(*TERMINAL 880KF1 - EL2008 ************************************************************************)
	qb880KF1_1_SignalToFockeReady								AT %Q* : BOOL; (* 880KF1_1 *)
	qb880KF1_5_SignalToFockeCutOut								AT %Q* : BOOL; (* 880KF1_5 *)
	qb880KF1_2_SignalToFockeRejectOuter							AT %Q* : BOOL; (* 880KF1_2 *)
	qb880KF1_6_SignalToFockeRejectLimitReachedTrigger			AT %Q* : BOOL; (* 880KF1_6 *)
	qb880KF1_3_SignalToFockeDynamicCameraTriggerPower			AT %Q* : BOOL; (* 880KF1_3 *)
	qb880KF1_7_Spare											AT %Q* : BOOL; (* 880KF1_7 *)
	qb880KF1_4_Spare											AT %Q* : BOOL; (* 880KF1_4 *)
	qb880KF1_8_Spare											AT %Q* : BOOL; (* 880KF1_8 *)

(*TERMINAL 881KF1 - EL2008 ************************************************************************)
	qb881KF1_1_MasterListCameraPower							AT %Q* : BOOL; (* 881KF1_1 *)
	qb881KF1_5_MasterListCameraTrigger							AT %Q* : BOOL; (* 881KF1_5 *)
	qb881KF1_2_AggregationCamera1Power							AT %Q* : BOOL; (* 881KF1_2 *)
	qb881KF1_6_AggregationCamera1Trigger						AT %Q* : BOOL; (* 881KF1_6 *)
	qb881KF1_3_AggregationCamera2Power							AT %Q* : BOOL; (* 881KF1_3 *)
	qb881KF1_7_AggregationCamera2Trigger						AT %Q* : BOOL; (* 881KF1_7 *)
	qb881KF1_4_AggregationCamera3Power							AT %Q* : BOOL; (* 881KF1_4 *)
	qb881KF1_8_AggregationCamera3Trigger						AT %Q* : BOOL; (* 881KF1_8 *)

(*TERMINAL 882KF1 - EL2008 ************************************************************************)
	qb882KF1_1_LightPoleGreen									AT %Q* : BOOL; (* 882KF1_1 *)
	qb882KF1_5_LightPoleAmber									AT %Q* : BOOL; (* 882KF1_5 *)
	qb882KF1_2_LightPoleRed										AT %Q* : BOOL; (* 882KF1_2 *)
	qb882KF1_6_LightPoleAlarm									AT %Q* : BOOL; (* 882KF1_6 *)
	qb882KF1_3_Spare											AT %Q* : BOOL; (* 882KF1_3 *)
	qb882KF1_7_Spare											AT %Q* : BOOL; (* 882KF1_7 *)
	qb882KF1_4_Spare											AT %Q* : BOOL; (* 882KF1_4 *)
	qb882KF1_8_Spare											AT %Q* : BOOL; (* 882KF1_8 *)
END_VAR

// ---- GVLs/Global Variables/InputsOutputs_CML/IOVariablesPAOL_CML.TcGVL
{attribute 'Tc2GvlVarNames'}
VAR_GLOBAL

(*METS TPD - PAOL (CML) *)
(*TERMINAL 546KF1 - EK1100 ******************************************************)

(*TERMINAL 547KF2 - EL4002 ******************************************************)

	qn547KF1_1_LightingIntensity						AT %Q* : INT; (*547KF1_1*)
	qn547KF1_2_Spare								AT %Q* : INT; (*547KF1_2*)

(*TERMINAL 560KF1 - EL1008 ******************************************************)
	ib560KF1_1_PrePackAggregationCameraRigTrigger		AT %I* : BOOL; (* 560KF1_1 *)
	ib560KF1_5_PackAggregationCamera1Trigger			AT %I* : BOOL; (* 560KF1_5 *)
	ib560KF1_2_PackAggregationCamera2Trigger			AT %I* : BOOL; (* 560KF1_2 *)
	ib560KF1_6_PackAggregationCamera3Trigger			AT %I* : BOOL; (* 560KF1_6 *)
	ib560KF1_3_PreMachineBuildBack					AT %I* : BOOL; (* 560KF1_3 *)
	ib560KF1_7_TPDExitBlock							AT %I* : BOOL; (* 560KF1_7 *)
	ib560KF1_4_ConveyorIndexContact					AT %I* : BOOL; (* 560KF1_4 *)		(*not used on C922 and C925 *)
	ib560KF1_8_PackIsolatorDrive						AT %I* : BOOL; (* 560KF1_8 *)

(*TERMINAL 5480KF1 - EL2008 ******************************************************)
	qb580KF1_1_PackAggregationCamera1Enable			AT %Q* : BOOL; (* 580KF1_1 *)
	qb580KF1_5_PackAggregationCamera2Enable			AT %Q* : BOOL; (* 580KF1_5 *)
	qb580KF1_2_PackAggregationCamera3Enable			AT %Q* : BOOL; (* 580KF1_2 *)
	qb580KF1_6_PackAggregationCamera1Power			AT %Q* : BOOL; (* 580KF1_6 *)
	qb580KF1_3_PackAggregationCamera2Power			AT %Q* : BOOL; (* 580KF1_3 *)
	qb580KF1_7_PackAggregationCamera3Power			AT %Q* : BOOL; (* 580KF1_7 *)
	qb580KF1_4_Spare								AT %Q* : BOOL; (* 580KF1_4 *)
	qb580KF1_8_PackCamerasLenseAir					AT %Q* : BOOL; (* 580KF1_8 *)

END_VAR

// ---- GVLs/Global Variables/InputsOutputs_CML/IOVariablesPLAS_CML.TcGVL
{attribute 'Tc2GvlVarNames'}
VAR_GLOBAL

(*TERMINAL XXXKF1 - EK1100 ******************************************************)


(*TERMINAL 747KF1 - EL4002 ******************************************************)
	qn747KF1_1_LightingIntensityPackAggregationCamera			AT %Q* : INT;
	qn747KF1_2_LightingIntensityPackConfirmationCamera			AT %Q* : INT;

(*TERMINAL 763KF1 - EL1008 ******************************************************)
	ib763KF1_1_MasterListCameraTrigSensor						AT %I* : BOOL;
	ib763KF1_5_SpareMasterListCameraTrigSensor					AT %I* : BOOL;		(* Option *)
	ib763KF1_2_AggregationCameraTrigSensor					AT %I* : BOOL;
	ib763KF1_6_SpareAggregationCamera1TrigSensor				AT %I* : BOOL;		(* Option *)
	ib763KF1_3_SpareAggregationCamera2TrigSensor				AT %I* : BOOL;		(* Option *)
	ib763KF1_7_PackQueueIndex								AT %I* : BOOL;
	ib763KF1_4_StackQueueIndex								AT %I* : BOOL; 		(* Option *)
	ib763KF1_8_SpareIndex									AT %I* : BOOL;		(* Option *)

(*TERMINAL 764KF1 - EL1008 ******************************************************)
	ib764KF1_1_OuterIndexComplete							AT %I* : BOOL;
	ib764KF1_5_SpareCameraTrigSensor							AT %I* : BOOL;		(* Option *)
	ib764KF1_2_Guard1 										AT %I* : BOOL;		(*FOCKE/GD Master list guard*)
	ib764KF1_6_Guard2										AT %I* : BOOL;		(*FOCKE/GD Master list guard*)
	ib764KF1_3_Guard3 										AT %I* : BOOL;		(*FOCKE/GD Aggregation guard*)
	ib764KF1_7_Guard4 										AT %I* : BOOL;		(*FOCKE/GD Aggregationt guard*) (*Option*)
	ib764KF1_4_OuterBrushOpen								AT %I* : BOOL;		(*Option*)
	ib764KF1_8_RejectTowerActive								AT %I* : BOOL;

(*TERMINAL 765KF1 (EL1008 8Ch. Dig. Input 24V, 3ms) ******************************************************)
	ib765KF1_1_FilmInPosition								AT %I*: BOOL;		(*Option*)
	ib765KF1_5_SparePrinterTrigger							AT %I*: BOOL;		(*Option*)
	ib765KF1_2_IntermediateCamera1TrigSesnor					AT %I*: BOOL;
	ib765KF1_6_HeatTunenelPackReject							AT %I*: BOOL;												(*not used on C922 and C925 *)
	ib765KF1_3_OuterAtAdditionalConveyor01 					AT %I*: BOOL;												(*not used on C922 and C925 *)
	ib765KF1_7_IntermediateCamera2TrigSesnor					AT %I*: BOOL;												(*not used on C922 and C925 *)
	ib765KF1_4_OuterAtReject								AT %I*: BOOL;		(*AdditionalConveyor01*)					(*not used on C922 and C925 *)
	ib765KF1_8_RejectConfirmation	 						AT %I*: BOOL;		(*AdditionalConveyor01*)					(*not used on C922 and C925 *)

(*TERMINAL 783KF1 - EL2008 ******************************************************)
	qb783KF1_1_MasterListCameraPower						AT %Q* : BOOL;
	qb783KF1_5_SpareMasterListCameraPower					AT %Q* : BOOL;		(* Option *)
	qb783KF1_2_SpareAggregationCameraPower					AT %Q* : BOOL;		(* Option *)
	qb783KF1_6_AggregationCamera1Power						AT %Q* : BOOL;
	qb783KF1_3_AggregationCamera2Power						AT %Q* : BOOL;
	qb783KF1_7_ConfirmationCamera1Power						AT %Q* : BOOL;
	qb783KF1_4_ConfirmationCamera2Power						AT %Q* : BOOL; 	(* Option *)
	qb783KF1_8_PLCControlledPackAggCamLightning			AT %Q* : BOOL;

(*TERMINAL 784KF1 - EL2008 ******************************************************)
	qb784KF1_1_MasterListCameraTrigger						AT %Q* : BOOL;
	qb784KF1_5_SpareMasterListCameraTrigger					AT %Q* : BOOL;		(* Option *)
	qb784KF1_2_AggregationCameraTrigger						AT %Q* : BOOL;
	qb784KF1_6_AggregationCamera1Trigger						AT %Q* : BOOL; 	(* Option *)
	qb784KF1_3_AggregationCamera2Trigger						AT %Q* : BOOL; 	(* Option *)
	qb784KF1_7_ConfirmationCamera1Trigger					AT %Q* : BOOL;
	qb784KF1_4_ConfirmationCamera2Trigger					AT %Q* : BOOL; 	(* Option *)
	qb784KF1_8_PLCControlledPackConfirmCamLightning		AT %Q* : BOOL;

(*TERMINAL 785KF1 (EL2008 8Ch. Dig. Output 24V, 3ms) ******************************************************)
	qb785KF1_1_IntermediateCamera1Trigger					AT %Q*: BOOL;
	qb785KF1_5_IntermediateCamera1Power					AT %Q*: BOOL;
	qb785KF1_2_IntermediateCamera2Trigger					AT %Q*: BOOL;												(*not used on C922 and C925 *)
	qb785KF1_6_IntermediateCamera3Power					AT %Q*: BOOL;												(*not used on C922 and C925 *)
	qb785KF1_3_RejectCylinderExtended						AT %Q*: BOOL;			(*AdditionalConveyor01*)				(*not used on C922 and C925 *)
	qb785KF1_7_RjectCylinderRetracted							AT %Q*: BOOL;			(*AdditionalConveyor01*)				(*not used on C922 and C925 *)
	qb785KF1_4_IntermediateCamera3Trigger					AT %Q*: BOOL;												(*not used on C922 and C925 *)
	qb785KF1_8_IntermediateCamera3Power					AT %Q*: BOOL;												(*not used on C922 and C925 *)

END_VAR

// ---- GVLs/Global Variables/InputsOutputs_OC/IOVariablesCX_OC.TcGVL
{attribute 'Tc2GvlVarNames'}
VAR_GLOBAL
(***************************Terminal States Diagnostic*****************************************************)

	istEtherCATMasterState							AT	%I*	: ST_CX_EtherCATMasterState;
	iaEtherCATSlaveState							AT 	%I*	: ARRAY [0..cMAX_ETHERCAT_SLAVES] OF UINT;

(*****************************Input/Output Cards*********************************************************)

	(*TERMINAL 45KF2 (EK1200-5000 EtherCAT Power supply (2A E-Bus)) ***************************************)

	(*TERMINAL 50KF1 (EL6001 Interface (RS232))  ********1-Channel Serial Interface RS232***********************)
	ib50A1_EL6001PortNo								AT %I* :  UINT;
	ist50A1_HandScannerCOMPortDataIn				AT %I* :  EL6InData22B;
	qst50A1_HandScannerCOMPortDataOut				AT %Q*: EL6OutData22B;

	(*TERMINAL 60KF1 (EL1008 8Ch. Dig. Input 24V, 3ms) ******************************************************)
	ib60KF1_1_Spare 								AT %I*: BOOL;
	ib60KF1_5_Spare									AT %I*: BOOL;
	ib60KF1_2_Spare									AT %I*: BOOL;
	ib60KF1_6_Spare									AT %I*: BOOL;
	ib60KF1_3_Spare 								AT %I*: BOOL;
	ib60KF1_7_Spare									AT %I*: BOOL;
	ib60KF1_4_Spare									AT %I*: BOOL;
	ib60KF1_8_Spare 	 							AT %I*: BOOL;

	(*TERMINAL 61KF1 (EL1008 8Ch. Dig. Input 24V, 3ms) ******************************************************)
	ib61KF1_1_DoorOpenZone1_SFCP					AT %I*: BOOL;
	ib61KF1_5_DoorOpenZone2_SFCP					AT %I*: BOOL;
	ib61KF1_2_CasePackerAutoRun_SFCP  				AT %I*: BOOL;
	ib61KF1_6_CaseRejected_SFCP		 				AT %I*: BOOL;
	ib61KF1_3_RowComplete_SFCP  					AT %I*: BOOL;
	ib61KF1_7_LayerComplete_SFCP  					AT %I*: BOOL;
	ib61KF1_4_CaseComplete_SFCP  					AT %I*: BOOL;
	ib61KF1_8_CaseDischarged_SFCP  					AT %I*: BOOL;

	(*TERMINAL 62KF1 (EL1008 8Ch. Dig. Input 24V, 3ms) ******************************************************)
	ib62KF1_1_CasePresentPosition01_SFCP								AT %I*: BOOL;
	ib62KF1_5_CasePresentPosition02_SFCP								AT %I*: BOOL;
	ib62KF1_2_CasePresentPosition03_SFCP						AT %I*: BOOL;
	ib62KF1_6_CasePresentPosition04_SFCP							AT %I*: BOOL;
	ib62KF1_3_CasePresentPosition05_SFCP							AT %I*: BOOL;
	ib62KF1_7_CasePresentPosition06_SFCP							AT %I*: BOOL;
	ib62KF1_4_CasePresentPosition07_SFCP								AT %I*: BOOL;
	ib62KF1_8_CasePresentPosition08_SFCP							AT %I*: BOOL;

	(*TERMINAL 63KF1 (EL1008 8Ch. Dig. Input 24V, 3ms) ******************************************************)
	ib63KF1_1_24VPowerSupplyOK 						AT %I*: BOOL;
	ib63KF1_5_EthernetSwitchOK 						AT %I*: BOOL;	 (* Option *)
	ib63KF1_2_CaseLabelValidationTrig_SFCP 			AT %I*: BOOL;
	ib63KF1_6_QAButtonRejectOuter_SFCP 				AT %I*: BOOL;
	ib63KF1_3_IntermediatePush_SFCP 				AT %I*: BOOL;
	ib63KF1_7_24VPowerSupplyAdditionalUnitOK			AT %I*: BOOL;
	ib63KF1_4_CasePresentPrintAreaSensor			AT %I*: BOOL;	 (* Option *)
	ib63KF1_8_CaseLeavingPrintAreaSensor			AT %I*: BOOL;	 (* Option *)

	(*TERMINAL 64KF1 (EL1008 8Ch. Dig. Input 24V, 3ms) ******************************************************)
	ib64KF1_1_PackSeparationDriveOK					AT %I*: BOOL;
	ib64KF1_5_Spare							AT %I*: BOOL;	(*  *)
	ib64KF1_2_IntermediateCameraTrigSesnorOK						AT %I*: BOOL;	(*  *)
	ib64KF1_6_AdditionalConveyorPlugConnected					AT %I*: BOOL;	(*  *)
	ib64KF1_3_OutfeedConveyorPlugConnected			AT %I*: BOOL; (**)
	ib64KF1_7_TransferConveyorPlugConnected			AT %I*: BOOL;	(* *)
	ib64KF1_4_Guard1 								AT %I*: BOOL; 	(* *)
	ib64KF1_8_Guard2								AT %I*: BOOL; 	(**)

	(*TERMINAL 65KF1 (EL1008 8Ch. Dig. Input 24V, 3ms) ******************************************************)
	ib65KF1_1_PSRisReset							AT %I*: BOOL;
	ib65KF1_5_PSRisOK								AT %I*: BOOL;
	ib65KF1_2_EmergencyStopFromPSR					AT %I*: BOOL;
	ib65KF1_6_EmergencyCircuitFromPSR 				AT %I*: BOOL;
	ib65KF1_3_AirDumpStatus					AT %I*: BOOL; 	(*  *)
	ib65KF1_7_Guard3								AT %I*: BOOL; 	(*  *)
	ib65KF1_4_Guard4								AT %I*: BOOL; 	(*   *)
	ib65KF1_8_Guard5								AT %I*: BOOL; 	(*  *)

	(*TERMINAL 66KF1 (EL1008 8Ch. Dig. Input 24V, 3ms) ******************************************************)
	ib66KF1_1_AirSupplyOK									AT %I*: BOOL;
	ib66KF1_5_PreMachineInAutorun					AT %I*: BOOL;		(*coneccted - input in PreMachine plug 18DX1 *)
	ib66KF1_2_PostMachineInAutorun					AT %I*: BOOL;		(*not coneccted - input in Safety plug 18DX2 *)
	ib66KF1_6_OuterRejectConfirmation				AT %I*: BOOL;		(*Duplicated*)
	ib66KF1_3_MainConveyorStart						AT %I*: BOOL;
	ib66KF1_7_CaseRejctConfirmCameraInReadCycle	AT %I*: BOOL;
	ib66KF1_4_CaseRejctConfirmCameraNoRead		AT %I*: BOOL;
	ib66KF1_8_CaseRejctConfirmCameraGoodRead		AT %I*: BOOL;

	(*TERMINAL 67KF1 (EL1008 8Ch. Dig. Input 24V, 3ms) ******************************************************)
	ib67KF1_1_Spare									AT %I*: BOOL;
	ib67KF1_5_Spare									AT %I*: BOOL;
	ib67KF1_2_Spare									AT %I*: BOOL;
	ib67KF1_6_Spare									AT %I*: BOOL;
	ib67KF1_3_Spare									AT %I*: BOOL;
	ib67KF1_7_Spare									AT %I*: BOOL;
	ib67KF1_4_Spare									AT %I*: BOOL;
	ib67KF1_8_Spare									AT %I*: BOOL;

	(*TERMINAL 69KF1 (EL1008 8Ch. Dig. Input 24V, 3ms) ******************************************************)
	ib69KF1_1_Labeller01Ready							AT %I*: BOOL;
	ib69KF1_5_Labeller01DataReady						AT %I*: BOOL;
	ib69KF1_2_Labeller01HomePosition							AT %I*: BOOL;
	ib69KF1_6_Labeller01LabelPrinted							AT %I*: BOOL;
	ib69KF1_3_Labeller01SummaryWarning							AT %I*: BOOL;
	ib69KF1_7_Labeller01Error								AT %I*: BOOL;
	ib69KF1_4_Labeller01AirPressureOK							AT %I*: BOOL;
	ib69KF1_8_Labeller01InPosition						AT %I*: BOOL;

	(*TERMINAL 70KF1 (EL1008 8Ch. Dig. Input 24V, 3ms) ******************************************************)
	ib70KF1_1_MainsSupplyHealthy					AT %I*: BOOL;	(*  *)
	ib70KF1_5_UPSHealthy							AT %I*: BOOL;	(*  *)
	ib70KF1_2_UPSBatteryMode						AT %I*: BOOL;	(*  *)
	ib70KF1_6_UPSBatteryCharging					AT %I*: BOOL;	(*  *)
	ib70KF1_3_Spare									AT %I*: BOOL; (**)
	ib70KF1_7_Spare								AT %I*: BOOL;	(* *)
	ib70KF1_4_Spare 								AT %I*: BOOL; 	(* *)
	ib70KF1_8_Spare								AT %I*: BOOL; 	(* *)

	(*TERMINAL 80KF1 (EL2008 8Ch. Dig. Output 24V, 0.5A) ******************************************************)
	qb80KF1_1_LightPoleGREEN  						AT %Q*: BOOL;
	qb80KF1_5_LightPoleAMBER  						AT %Q*: BOOL;
	qb80KF1_2_LightPoleRED  						AT %Q*: BOOL;
	qb80KF1_6_LightPoleALARM  						AT %Q*: BOOL;	 (* Option *)
	qb80KF1_3_LightHandscannerBoxGreen 				AT %Q*: BOOL;	 (* Option *)
	qb80KF1_7_LightHandscannerBoxRed  				AT %Q*: BOOL;	 (* Option *)
	qb80KF1_4_Spare  								AT %Q*: BOOL;
	qb80KF1_8_OuterRejectSignal   					AT %Q*: BOOL;	 (*Option*)

	(*TERMINAL 81KF1 (EL2008 8Ch. Dig. Output 24V, 0.5A) ******************************************************)
	qb81KF1_1_SafetyReset	  						AT %Q*: BOOL;
	qb81KF1_5_PackSeperationDriveFaultAck			AT %Q*: BOOL;
	qb81KF1_2_PackSeperationDriveBrakeRelease		AT %Q*: BOOL;	 (* Option *)
	qb81KF1_6_CaseRejctConfirmCameraPower 								AT %Q*: BOOL;
	qb81KF1_3_CaseRejctConfirmCameraTrigger									AT %Q*: BOOL;
	qb81KF1_7_PreMachineAddditionalCutOut			AT %Q*: BOOL;	 (* not coneccted - output in Safety plug 18DX1  *)
	qb81KF1_4_PreMachineCutOut						AT %Q*: BOOL;	(*coneccted - output in PreMachine plug 18DX1 *)
	qb81KF1_8_PostMachineAddditionalCutOut	 					AT %Q*: BOOL;		(* not coneccted - output in PostMachine Safety plug 18DX2 *)

	(*TERMINAL 82KF1 (EL2008 8Ch. Dig. Output 24V, 0.5A) ******************************************************)
	qb82KF1_1_PostMachineCutOut_STCP		  					AT %Q*: BOOL;		(*coneccted - output in PostMachine plug 19DX2 *)
	qb82KF1_5_CaseValidationOK_STCP					AT %Q*: BOOL;
	qb82KF1_2_OuterValidationOK_STCP 				AT %Q*: BOOL;
	qb82KF1_6_CaseContentOK_STCP					AT %Q*: BOOL;
	qb82KF1_3_LabellerInhibit_STL					AT %Q*: BOOL;
	qb82KF1_7_RejectSignal3_STL 					AT %Q*: BOOL;	(*  *)
	qb82KF1_4_Miscellaneous_STL						AT %Q*: BOOL;	(*  *)
	qb82KF1_8_Spare			 						AT %Q*: BOOL;

	(*TERMINAL 83KF1 (EL2008 8Ch. Dig. Output 24V, 0.5A) ******************************************************)
	qb83KF1_1_PackSepparationDriveRun									AT %Q*: BOOL;
	qb83KF1_5_AdditionalConveyor01Run									AT %Q*: BOOL;
	qb83KF1_2_AdditionalConveyor02Run									AT %Q*: BOOL;
	qb83KF1_6_Spare									AT %Q*: BOOL;
	qb83KF1_3_Spare									AT %Q*: BOOL;
	qb83KF1_7_Spare									AT %Q*: BOOL;
	qb83KF1_4_Spare									AT %Q*: BOOL;
	qb83KF1_8_Labeller01DoorGuardOpen			AT %Q*: BOOL;

	(*TERMINAL 84KF1 (EL2008 8Ch. Dig. Output 24V, 0.5A) ******************************************************)
	qb84KF1_1_Spare								AT %Q*: BOOL;
	qb84KF1_5_Spare									AT %Q*: BOOL;
	qb84KF1_2_Spare									AT %Q*: BOOL;
	qb84KF1_6_Spare									AT %Q*: BOOL;
	qb84KF1_3_Spare									AT %Q*: BOOL;
	qb84KF1_7_Spare									AT %Q*: BOOL;
	qb84KF1_4_Spare									AT %Q*: BOOL;
	qb84KF1_8_Spare									AT %Q*: BOOL;

	(*TERMINAL 88KF1 (EL4002 2Ch. Analog Output, 0…10 V, 12 bit) ******************************************************)
	qn88KF1_1_PackSeparationDriveCh1							AT %Q* : INT;
	qn88KF1_2_Spare											AT %Q* : INT;

	(*TERMINAL 90KF1 (EL2624 4Ch. Relay Output, 125 V AC, 30 V DC, 0.5 A AC, 2 A DC)******************)
	qb90KF1_1_Labeller01ResetSignal					AT %Q*: BOOL;		(**)
	qb90KF1_2_Labeller01PrintSignal							AT %Q*: BOOL;		(**)
	qb90KF1_3_Labeller01ApplySignal1						AT %Q*: BOOL;		(**)
	qb90KF1_4_Labeller01ApplySignal2										AT %Q*: BOOL;

	(*TERMINAL 97KF1 - EL6631 -  PROFINET IO Controller ********************************************************)
	ist97KF1_Master01PNetState 						AT %I* : ST_CX_EtherCATMasterPNetState;

	(*DRIVE  3T1  - G120C ************************************************************************************)
	ist3T1_outerseparation							AT %I* : ST_DRIVE_INPUT;
	qst3T1_outerseparation							AT %Q* : ST_DRIVE_OUTPUT;

	(*DRIVE  4T1  - G120C ************************************************************************************)
	ist4T1_transferconveyor							AT %I* : ST_DRIVE_INPUT;
	qst4T1_transferconveyor							AT %Q* : ST_DRIVE_OUTPUT;

	(*DRIVE  5T1  - G120C ************************************************************************************)
	ist5T1_outfeedconveyor							AT %I* : ST_DRIVE_INPUT;
	qst5T1_outfeedconveyor							AT %Q* : ST_DRIVE_OUTPUT;

	(*DRIVE  6T1  - G120C ************************************************************************************)
	ist6T1_additionalconveyor						AT %I* : ST_DRIVE_INPUT;
	qst6T1_additionalconveyor					AT %Q* : ST_DRIVE_OUTPUT;
END_VAR

// ---- GVLs/Global Variables/InputsOutputs_OC/IOVariablesEUCA_OC.TcGVL
{attribute 'Tc2GvlVarNames'}
VAR_GLOBAL

(*TERMINAL XXXKF1 - EK1100 **********************************************************)

(*TERMINAL 350KF1 (EL6001 Interface (RS232))  ********1-Channel Serial Interface RS232***********************)
	ib350A1_EL6001PortNo								AT %I* :  UINT;
	ist350A1_HandScannerCOMPortDataIn					AT %I* :  EL6InData22B;
	qst350A1_HandScannerCOMPortDataOut					AT %Q*: EL6OutData22B;

(*TERMINAL 351KF1 - EL4002 ******************************************************)
	qn351KF1_1_OuterValidationLightingIntensity			AT %Q* : INT;
	qn351KF1_2_OuterAggregationLightingIntensity		AT %Q* : INT;

(*TERMINAL 352KF1 - EL4002 ******************************************************)
	qn352KF1_1_CaseContentValidationLightingIntensity	AT %Q* : INT;
	qn352KF1_2_LightingIntensity							AT %Q* : INT;

(*TERMINAL 360KF1 - EL1008 ***********************************************************)
	ib360KF1_1_OuterAtInfeed							AT %I* : BOOL;	(* Option *)
	ib360KF1_5_OuterInfeedBlocked						AT %I* : BOOL;	(* Option clamp*)
	ib360KF1_2_OuterAtLabeller							AT %I* : BOOL;	(* Option gate*)
	ib360KF1_6_PackConfirmationCameraTrigSensor			AT %I* : BOOL;
	ib360KF1_3_OuterValidationCameraTrigSensor 					AT %I* : BOOL;
	ib360KF1_7_OuterAtReject							AT %I* : BOOL;
	ib360KF1_4_RejectConfirmation						AT %I* : BOOL;
	ib360KF1_8_RejectBinFull								AT %I* : BOOL;

(*TERMINAL 361KF1 - EL1008 ***********************************************************)
	ib361KF1_1_OuterClampExtended							AT %I* : BOOL;
	ib361KF1_5_OuterGateExtended					AT %I* : BOOL;
	ib361KF1_2_OuterGateRetracted						AT %I* : BOOL;
	ib361KF1_6_OuterGateImpactSensor						AT %I* : BOOL;
	ib361KF1_3_RejectCylinderExtended					AT %I* : BOOL;
	ib361KF1_7_RejectCylinderRetracted					AT %I* : BOOL;
	ib361KF1_4_EUCAExitBlocked										AT %I* : BOOL;	(* Option *)
	ib361KF1_8_EUCABuildBack									AT %I* : BOOL;

(*TERMINAL 362KF1 - EL1008 ************************************************************)
	ib362KF1_1_Labeller02Ready							AT %I*: BOOL;
	ib362KF1_5_Labeller02DataReady						AT %I*: BOOL;
	ib362KF1_2_Labeller02HomePosition 			AT %I*: BOOL;
	ib362KF1_6_Labeller02LabelPrinted						AT %I*: BOOL;
	ib362KF1_3_Labeller02SummaryWarning					AT %I*: BOOL;
	ib362KF1_7_Labeller02Error							AT %I*: BOOL;
	ib362KF1_4_Labeller02AirPressureOK							AT %I*: BOOL;
	ib362KF1_8_Labeller02InPosition					AT %I*: BOOL;	(* ??? *)

(*TERMINAL 363KF1 (EL1008 8Ch. Dig. Input 24V, 3ms) ***************************************)
	ib363KF1_1_QAButtonRejectOuter						AT %I*: BOOL;	(* Option *)
	ib363KF1_5_IntermediatePushSensor					AT %I*: BOOL;
	ib363KF1_2_CaseLabelValidationCameraTrigSensor 		AT %I*: BOOL;
	ib363KF1_6_OuterAggregationCameraTrigSensor			AT %I*: BOOL;	(* *)
	ib363KF1_3_RowCompleteSensor						AT %I*: BOOL;
	ib363KF1_7_LayerCompleteSensor						AT %I*: BOOL;
	ib363KF1_4_CaseCompleteSensor						AT %I*: BOOL;
	ib363KF1_8_CaseDischargedSensor						AT %I*: BOOL;

(*TERMINAL 366KF1 (EL1008 8Ch. Dig. Input 24V, 3ms) ****************************************)
	ib366KF1_1_OuterAtAdditionalConveyor02									AT %I*: BOOL;
	ib366KF1_5_ExitBlockedAdditionalConveyor02									AT %I*: BOOL;
	ib366KF1_2_Spare									AT %I*: BOOL;
	ib366KF1_6_Spare									AT %I*: BOOL;
	ib366KF1_3_Spare									AT %I*: BOOL;
	ib366KF1_7_Spare									AT %I*: BOOL;
	ib366KF1_4_Spare								AT %I*: BOOL;
	ib366KF1_8_RemoteAirSupplyOK									AT %I*: BOOL;

(*TERMINAL 380KF1 - EL2008 (EL2008 8Ch. Dig. Output 24V, 0.5A) ********************************)
	qb380KF1_1_ClampCylinderExtend				AT %Q*: BOOL;
	qb380KF1_5_Spare						 			AT %Q*: BOOL;
	qb380KF1_2_GateCylinderExtend 						AT %Q*: BOOL;		(**)
	qb380KF1_6_GateCylinderRetract	 					AT %Q*: BOOL;		(**)
	qb380KF1_3_RejectCylinderExtend						AT %Q*: BOOL;
	qb380KF1_7_RejectCylinderRetract			  		AT %Q*: BOOL;
	qb380KF1_4_Spare								AT %Q*: BOOL;
	qb380KF1_8_PLCControlledAggCameraLightning			AT %Q*: BOOL; (**)

(*TERMINAL 381KF1 (EL2008 8Ch. Dig. Output 24V, 0.5A) ***************************************)
	qb381KF1_1_RearConfirmationCameraTrigger			AT %Q*: BOOL;
	qb381KF1_5_RearConfirmationCameraPower				AT %Q*: BOOL;
	qb381KF1_2_FrontConfirmationCameraTrigger			AT %Q*: BOOL;
	qb381KF1_6_FrontConfirmationCameraPower	 			AT %Q*: BOOL;
	qb381KF1_3_OuterValidationCameraTrig 					AT %Q*: BOOL;
	qb381KF1_7_OuterValidationCameraPower				AT %Q*: BOOL;
	qb381KF1_4_OuterAggregationCameraTrig					AT %Q*: BOOL;
	qb381KF1_8_OuterAggregationCameraPower					AT %Q*: BOOL;

(*TERMINAL 382KF1 (EL2008 8Ch. Dig. Output 24V, 0.5A) ****************************************)
	qb382KF1_1_CaseContentValidationCameraTrig				AT %Q*: BOOL;
	qb382KF1_5_CaseContentValidationCameraPower			AT %Q*: BOOL;
	qb382KF1_2_CaseLabelValidationCameraTrig				AT %Q*: BOOL;
	qb382KF1_6_CaseLabelValidationCameraPower	 			AT %Q*: BOOL;
	qb382KF1_3_OuterValidationCameraLightning					AT %Q*: BOOL;		(**)
	qb382KF1_7_OuterAggregationCameraLightning				AT %Q*: BOOL;		(**)
	qb382KF1_4_CaseContentValidationCameraLightning			AT %Q*: BOOL;		(**)
	qb382KF1_8_Labeller02DoorGuardOpen				AT %Q*: BOOL;		(**)

(*TERMINAL 390KF1 (EL2624 4Ch. Relay Output, 125 V AC, 30 V DC, 0.5 A AC, 2 A DC)******************)
	qb390KF1_1_Labeller02ResetSignal						AT %Q*: BOOL;
	qb390KF1_2_Labeller02PrintSignal						AT %Q*: BOOL;
	qb390KF1_3_Labeller02ApplySignal1						AT %Q*: BOOL;
	qb390KF1_4_Labeller02ApplySignal2								AT %Q*: BOOL;

END_VAR

// ---- GVLs/Global Variables/InputsOutputs_OC/IOVariablesPAOL_OC.TcGVL
{attribute 'Tc2GvlVarNames'}
VAR_GLOBAL

(*TERMINAL XXXKF1 - EK1100 ******************************************************)

(*TERMINAL 647KF1 - EL4002 ******************************************************)
	qn647KF1_1_LightingIntensity							AT %Q* : INT;
	qn647KF1_2_Spare									AT %Q* : INT;

(*TERMINAL 660KF1 - EL1008 ******************************************************)
	ib660KF1_1_PackAggregationCameraRigTrigger			AT %I* : BOOL;
	ib660KF1_5_PackAggregationCamera1Trigger				AT %I* : BOOL;
	ib660KF1_2_PackAggregationCamera2Trigger				AT %I* : BOOL;
	ib660KF1_6_PackAggregationCamera3Trigger				AT %I* : BOOL;
	ib660KF1_3_PreMachineBuildBack						AT %I* : BOOL;
	ib660KF1_7_TPDExitBlock								AT %I* : BOOL;
	ib660KF1_4_PackAggregationCamera4Trigger				AT %I* : BOOL;	(* Option *)
	ib660KF1_8_PackIsolatorDrive							AT %I* : BOOL;

(*TERMINAL 680KF1 - EL2008 ******************************************************)
	qb680KF1_1_PackAggregationCamera1Enable				AT %Q* : BOOL;
	qb680KF1_5_PackAggregationCamera2Enable				AT %Q* : BOOL;
	qb680KF1_2_PackAggregationCamera3Enable				AT %Q* : BOOL;
	qb680KF1_6_PackAggregationCamera1Power				AT %Q* : BOOL;
	qb680KF1_3_PackAggregationCamera2Power				AT %Q* : BOOL;
	qb680KF1_7_PackAggregationCamera3Power				AT %Q* : BOOL;
	qb680KF1_4_PackAggregationCamera4Enable				AT %Q* : BOOL;
	qb680KF1_8_PackCamerasLenseAir						AT %Q* : BOOL;

END_VAR

// ---- GVLs/Global Variables/InputsOutputs_OC/IOVariablesPLAS_OC.TcGVL
{attribute 'Tc2GvlVarNames'}
VAR_GLOBAL

(*TERMINAL XXXKF1 - EK1100 ******************************************************)


(*TERMINAL 747KF1 - EL4002 ******************************************************)
	qn747KF1_1_LightingIntensityPackAggregationCamera							AT %Q* : INT;
	qn747KF1_2_LightingIntensityPackConfirmationCamera							AT %Q* : INT;

(*TERMINAL 748KF1 - EL4002 ******************************************************)
	qn748KF1_1_LightingIntensityMasterListCamera		AT %Q* : INT;
	qn748KF1_2_Spare										AT %Q* : INT;

(*TERMINAL 763KF1 - EL1008 ******************************************************)
	ib763KF1_1_MasterListCameraTrigSensor					AT %I* : BOOL;
	ib763KF1_5_SpareMasterListCameraTrigSensor			AT %I* : BOOL;		(* Option *)
	ib763KF1_2_AggregationCameraTrigSensor				AT %I* : BOOL;
	ib763KF1_6_SpareAggregationCamera1TrigSensor		AT %I* : BOOL;		(* Option *)
	ib763KF1_3_SpareAggregationCamera2TrigSensor		AT %I* : BOOL;		(* Option *)
	ib763KF1_7_PackQueueIndex								AT %I* : BOOL; 		(* Option *)
	ib763KF1_4_StackQueueIndex								AT %I* : BOOL; 		(* Option *)
	ib763KF1_8_SpareIndex											AT %I* : BOOL;

(*TERMINAL 764KF1 - EL1008 ******************************************************)
	ib764KF1_1_OuterIndexComplete							AT %I* : BOOL;
	ib764KF1_5_SpareCameraTrigSesnor						AT %I* : BOOL;		(* Option *)
	ib764KF1_2_Guard1 										AT %I* : BOOL;		(*FOCKE/GD Master list guard*)
	ib764KF1_6_Guard2										AT %I* : BOOL;		(*FOCKE/GD Master list guard*)
	ib764KF1_3_Guard3 										AT %I* : BOOL;		(*FOCKE/GD Aggregation guard*)
	ib764KF1_7_Guard4 										AT %I* : BOOL;		(*FOCKE/GD Aggregationt guard*)
	ib764KF1_4_OuterBrushOpen								AT %I* : BOOL;
	ib764KF1_8_RejectTowerActive							AT %I* : BOOL;

(*TERMINAL 765KF1 (EL1008 8Ch. Dig. Input 24V, 3ms) ******************************************************)
	ib765KF1_1_FilmInPosition 								AT %I*: BOOL;
	ib765KF1_5_SparePrinterTrigger							AT %I*: BOOL;
	ib765KF1_2_IntermediateCamera1TrigSesnor				AT %I*: BOOL;
	ib765KF1_6_HeatTunelPackReject							AT %I*: BOOL;
	ib765KF1_3_OuterAtAdditionalConveyor01 				AT %I*: BOOL;
	ib765KF1_7_IntermediateCamera2TrigSesnor				AT %I*: BOOL;
	ib765KF1_4_OuterAtReject									AT %I*: BOOL;		(*AdditionalConveyor01*)
	ib765KF1_8_RejectConfirmation	 						AT %I*: BOOL;		(*AdditionalConveyor01*)

(*TERMINAL 766KF1 - EL1008 ******************************************************)
	ib766KF1_1_RejectCylinderExtended						AT %I* : BOOL;
	ib766KF1_5_RejectCylinderRetracted						AT %I* : BOOL;		(*  *)
	ib766KF1_2_RejectBinFull 									AT %I* : BOOL;		(*AdditionalConveyor01*)
	ib766KF1_6_ExitBlockedAdditionalConveyor01				AT %I* : BOOL;
	ib766KF1_3_IntermediateCamera3TrigSesnor				AT %I* : BOOL;
	ib766KF1_7_Spare											AT %I* : BOOL;	(*Potentially for GD Additional Master list guard*)
	ib766KF1_4_Spare											AT %I* : BOOL;		(* Guard5 Potentially for GD Wrapper door*)
	ib766KF1_8_Spare											AT %I* : BOOL;			(* Guard6 Potentially for GD Wrapper door*)

(*TERMINAL 767KF1 - EL1008 ******************************************************)
	ib767KF1_1_ConveyorInterfaceInputSignal1				AT %I* : BOOL;
	ib767KF1_5_ConveyorInterfaceInputSignal2				AT %I* : BOOL;		(*  *)
	ib767KF1_2_RejectTower2Active							AT %I* : BOOL;		(**)
	ib767KF1_6_Spare											AT %I* : BOOL;
	ib767KF1_3_Spare											AT %I* : BOOL;
	ib767KF1_7_Spare 											AT %I* : BOOL;
	ib767KF1_4_Spare											AT %I* : BOOL;
	ib767KF1_8_Spare											AT %I* : BOOL;


(*TERMINAL 783KF1 - EL2008 ******************************************************)
	qb783KF1_1_MasterListCameraPower						AT %Q* : BOOL;
	qb783KF1_5_SpareMasterListCameraPower					AT %Q* : BOOL;	(* Option *)
	qb783KF1_2_SpareAggregationCameraPower				AT %Q* : BOOL;	(* Option *)
	qb783KF1_6_AggregationCamera1Power					AT %Q* : BOOL;
	qb783KF1_3_AggregationCamera2Power					AT %Q* : BOOL;
	qb783KF1_7_ConfirmationCamera1Power					AT %Q* : BOOL; 	(* Option *)
	qb783KF1_4_ConfirmationCamera2Power					AT %Q* : BOOL; 	(* Option *)
	qb783KF1_8_PLCControlledAggCamerasLightning			AT %Q* : BOOL;

(*TERMINAL 784KF1 - EL2008 ******************************************************)
	qb784KF1_1_MasterListCameraTrigger						AT %Q* : BOOL;
	qb784KF1_5_SpareMasterListCameraTrigger				AT %Q* : BOOL;	(* Option *)
	qb784KF1_2_AggregationCameraTrigger					AT %Q* : BOOL;
	qb784KF1_6_SpareAggregationCamera1Trigger			AT %Q* : BOOL; 	(* Option *)
	qb784KF1_3_SpareAggregationCamera2Trigger			AT %Q* : BOOL; 	(* Option *)
	qb784KF1_7_ConfirmationCamera1Trigger					AT %Q* : BOOL; 	(* Option *)
	qb784KF1_4_ConfirmationCamera2Trigger					AT %Q* : BOOL; 	(* Option *)
	qb784KF1_8_PLCControlledConfCameraLightning			AT %Q* : BOOL;

(*TERMINAL 785KF1 (EL2008 8Ch. Dig. Output 24V, 3ms) ******************************************************)
	qb785KF1_1_IntermediateCamera1Trigger					AT %Q*: BOOL;
	qb785KF1_5_IntermediateCamera1Power					AT %Q*: BOOL;
	qb785KF1_2_IntermediateCamera2Trigger					AT %Q*: BOOL;
	qb785KF1_6_IntermediateCamera3Power					AT %Q*: BOOL;
	qb785KF1_3_RejectCylinderExtended						AT %Q*: BOOL;			(*AdditionalConveyor01*)
	qb785KF1_7_RjectCylinderRetracted						AT %Q*: BOOL;			(*AdditionalConveyor01*)
	qb785KF1_4_IntermediateCamera3Trigger					AT %Q*: BOOL;
	qb785KF1_8_IntermediateCamera3Power					AT %Q*: BOOL;

(*TERMINAL 786KF1 - EL2008 ******************************************************)
	qb786KF1_1_ConveyorInterfaceOutputSignal1				AT %Q* : BOOL;
	qb786KF1_5_ConveyorInterfaceOutputSignal2				AT %Q* : BOOL;	(* Option *)
	qb786KF1_2_Spare											AT %Q* : BOOL;	(* Option *)
	qb786KF1_6_Spare											AT %Q* : BOOL;
	qb786KF1_3_Spare											AT %Q* : BOOL;
	qb786KF1_7_Spare											AT %Q* : BOOL; 	(* Option *)
	qb786KF1_4_Spare											AT %Q* : BOOL; 	(* Option *)
	qb786KF1_8_PLCControlledMLCamerasLightning			AT %Q* : BOOL;

END_VAR

// ---- GVLs/Global Variables/InputsOutputs_SFLX/IOVariablesCX_SFLX.TcGVL
{attribute 'Tc2GvlVarNames'}
VAR_GLOBAL
(***************************Terminal States Diagnostic*****************************************************)

	istEtherCATMasterState							AT	%I*	: ST_CX_EtherCATMasterState;
	iaEtherCATSlaveState							AT 	%I*	: ARRAY [0..cMAX_ETHERCAT_SLAVES] OF UINT;

(*****************************Input/Output Cards*********************************************************)

	(*TERMINAL 45KF2 (EK1200-5000 EtherCAT Power supply (2A E-Bus)) ***************************************)

	(*TERMINAL 50KF1 (EL6001 Interface (RS232))  ********1-Channel Serial Interface RS232***********************)
	ib50A1_EL6001PortNo								AT %I* :  UINT;
	ist50A1_HandScannerCOMPortDataIn				AT %I* :  EL6InData22B;
	qst50A1_HandScannerCOMPortDataOut				AT %Q*: EL6OutData22B;

	(*TERMINAL 60KF1 (EL1008 8Ch. Dig. Input 24V, 3ms) ******************************************************)
	ib60KF1_1_Spare 								AT %I*: BOOL;
	ib60KF1_5_Spare									AT %I*: BOOL;
	ib60KF1_2_Spare									AT %I*: BOOL;
	ib60KF1_6_Spare									AT %I*: BOOL;
	ib60KF1_3_Spare 								AT %I*: BOOL;
	ib60KF1_7_Spare									AT %I*: BOOL;
	ib60KF1_4_Spare									AT %I*: BOOL;
	ib60KF1_8_Spare 	 							AT %I*: BOOL;

	(*TERMINAL 61KF1 (EL1008 8Ch. Dig. Input 24V, 3ms) ******************************************************)
	ib61KF1_1_DoorOpenZone1_SFCP					AT %I*: BOOL;
	ib61KF1_5_DoorOpenZone2_SFCP					AT %I*: BOOL;
	ib61KF1_2_CasePackerAutoRun_SFCP  				AT %I*: BOOL;
	ib61KF1_6_CaseRejected_SFCP		 				AT %I*: BOOL;
	ib61KF1_3_RowComplete_SFCP  					AT %I*: BOOL;
	ib61KF1_7_LayerComplete_SFCP  					AT %I*: BOOL;
	ib61KF1_4_CaseComplete_SFCP  					AT %I*: BOOL;
	ib61KF1_8_CaseDischarged_SFCP  					AT %I*: BOOL;

	(*TERMINAL 62KF1 (EL1008 8Ch. Dig. Input 24V, 3ms) ******************************************************)
	ib62KF1_1_Spare									AT %I*: BOOL;
	ib62KF1_5_Spare 								AT %I*: BOOL;
	ib62KF1_2_Spare 								AT %I*: BOOL;
	ib62KF1_6_Spare 								AT %I*: BOOL;
	ib62KF1_3_Spare									AT %I*: BOOL;
	ib62KF1_7_Spare 								AT %I*: BOOL;
	ib62KF1_4_Spare 								AT %I*: BOOL;
	ib62KF1_8_Spare 								AT %I*: BOOL;

	(*TERMINAL 63KF1 (EL1008 8Ch. Dig. Input 24V, 3ms) ******************************************************)
	ib63KF1_1_24VPowerSupplyOK 						AT %I*: BOOL;
	ib63KF1_5_EthernetSwitchOK 						AT %I*: BOOL;	 (* Option *)
	ib63KF1_2_CaseLabelValidationTrig_SFCP 			AT %I*: BOOL;
	ib63KF1_6_QAButtonRejectOuter_SFCP 				AT %I*: BOOL;
	ib63KF1_3_IntermediatePush_SFCP 				AT %I*: BOOL;
	ib63KF1_7_Spare									AT %I*: BOOL;
	ib63KF1_4_CasePresentPrintAreaSensor			AT %I*: BOOL;	 (* Option *)
	ib63KF1_8_CaseLeavingPrintAreaSensor			AT %I*: BOOL;	 (* Option *)

	(*TERMINAL 64KF1 (EL1008 8Ch. Dig. Input 24V, 3ms) ******************************************************)
	ib64KF1_1_MainsSupplyHealthy					AT %I*: BOOL;	(* UPS *)
	ib64KF1_5_UPSHealthy							AT %I*: BOOL;	(* UPS *)
	ib64KF1_2_UPSBatteryMode						AT %I*: BOOL;	(* UPS *)
	ib64KF1_6_UPSBatteryCharging					AT %I*: BOOL;	(* UPS *)
	ib64KF1_3_TransferConveyorPlugConnected			AT %I*: BOOL; (*LARS and SFLX*)
	ib64KF1_7_OutfeedConveyorPlugConnected			AT %I*: BOOL;	(* SFLX*)
	ib64KF1_4_Guard1 								AT %I*: BOOL; 	(* LARS Transfer Coveyor printer*)
	ib64KF1_8_Guard2								AT %I*: BOOL; 	(* LARS Transfer Coveyor or pinch guard*)

	(*TERMINAL 65KF1 (EL1008 8Ch. Dig. Input 24V, 3ms) ******************************************************)
	ib65KF1_1_PSRisReset							AT %I*: BOOL;
	ib65KF1_5_PSRisOK								AT %I*: BOOL;
	ib65KF1_2_EmergencyStopFromPSR					AT %I*: BOOL;
	ib65KF1_6_EmergencyCircuitFromPSR 				AT %I*: BOOL;
	ib65KF1_3_Guard6									AT %I*: BOOL; 	(*  SFLX*)
	ib65KF1_7_Guard3								AT %I*: BOOL; 	(*  SFLX*)
	ib65KF1_4_Guard4								AT %I*: BOOL; 	(*  SFLX *)
	ib65KF1_8_Guard5								AT %I*: BOOL; 	(*  SFLX*)

	(*TERMINAL 66KF1 (EL1008 8Ch. Dig. Input 24V, 3ms) ******************************************************)
	ib66KF1_1_Spare									AT %I*: BOOL;
	ib66KF1_5_PreMachineInAutorun					AT %I*: BOOL;		(*coneccted - input in PreMachine plug 18DX1 *)
	ib66KF1_2_PostMachineInAutorun					AT %I*: BOOL;		(*not coneccted - input in Safety plug 18DX2 *)
	ib66KF1_6_Spare									AT %I*: BOOL;
	ib66KF1_3_Spare									AT %I*: BOOL;
	ib66KF1_7_Spare									AT %I*: BOOL;
	ib66KF1_4_Spare									AT %I*: BOOL;
	ib66KF1_8_Spare									AT %I*: BOOL;

	(*TERMINAL 67KF1 (EL1008 8Ch. Dig. Input 24V, 3ms) ******************************************************)
	ib67KF1_1_Spare									AT %I*: BOOL;
	ib67KF1_5_Spare									AT %I*: BOOL;
	ib67KF1_2_Spare									AT %I*: BOOL;
	ib67KF1_6_Spare									AT %I*: BOOL;
	ib67KF1_3_Spare									AT %I*: BOOL;
	ib67KF1_7_Spare									AT %I*: BOOL;
	ib67KF1_4_Spare									AT %I*: BOOL;
	ib67KF1_8_Spare									AT %I*: BOOL;

	(*TERMINAL 68KF1 (EL1008 8Ch. Dig. Input 24V, 3ms) ******************************************************)
	ib68KF1_1_ReadyToPrint							AT %I*: BOOL;		(*M-Series Printer Ready*)
	ib68KF1_5_BufferNotEmpty						AT %I*: BOOL;		(*M-Series Data Ready*)
	ib68KF1_2_PrintDone								AT %I*: BOOL;		(*M-Series Label Printed*)
	ib68KF1_6_PrinterWarning							AT %I*: BOOL;		(*M-Series Summary Warningy*)
	ib68KF1_3_PrinterError							AT %I*: BOOL;		(*M-Series Summary Error*)
	ib68KF1_7_Spare									AT %I*: BOOL;
	ib68KF1_4_AdditionalConveyorPlugConnected	AT %I*: BOOL;
	ib68KF1_8_Spare									AT %I*: BOOL;

	(*TERMINAL 80KF1 (EL2008 8Ch. Dig. Output 24V, 0.5A) ******************************************************)
	qb80KF1_1_LightPoleGREEN  						AT %Q*: BOOL;
	qb80KF1_5_LightPoleAMBER  						AT %Q*: BOOL;
	qb80KF1_2_LightPoleRED  						AT %Q*: BOOL;
	qb80KF1_6_LightPoleALARM  						AT %Q*: BOOL;	 (* Option *)
	qb80KF1_3_LightHandscannerBoxGreen 				AT %Q*: BOOL;	 (* Option *)
	qb80KF1_7_LightHandscannerBoxRed  				AT %Q*: BOOL;	 (* Option *)
	qb80KF1_4_Spare  								AT %Q*: BOOL;
	qb80KF1_8_OuterRejectSignal   					AT %Q*: BOOL;	 (*Option nie uzywamy*)

	(*TERMINAL 81KF1 (EL2008 8Ch. Dig. Output 24V, 0.5A) ******************************************************)
	qb81KF1_1_SafetyReset	  						AT %Q*: BOOL;
	qb81KF1_5_Spare 								AT %Q*: BOOL;
	qb81KF1_2_PackSeperationDriveBrakeRelease		AT %Q*: BOOL;	 (* Option *)
	qb81KF1_6_Spare 								AT %Q*: BOOL;
	qb81KF1_3_Spare									AT %Q*: BOOL;
	qb81KF1_7_PreMachineAddditionalCutOut			AT %Q*: BOOL;	 (* Option *)
	qb81KF1_4_PreMachineCutOut						AT %Q*: BOOL;(*coneccted - output in PreMachine plug 18DX1 *)
	qb81KF1_8_PostMachineRun	 					AT %Q*: BOOL;		(* not coneccted - output in Safety plug 18DX2 *)

	(*TERMINAL 82KF1 (EL2008 8Ch. Dig. Output 24V, 0.5A) ******************************************************)
	qb82KF1_1_CutOut_STCP		  					AT %Q*: BOOL;
	qb82KF1_5_CaseValidationOK_STCP					AT %Q*: BOOL;
	qb82KF1_2_OuterValidationOK_STCP 				AT %Q*: BOOL;
	qb82KF1_6_CaseContentOK_STCP					AT %Q*: BOOL;
	qb82KF1_3_LabellerInhibit_STL					AT %Q*: BOOL;
	qb82KF1_7_RejectSignal3_STL 					AT %Q*: BOOL;	(* Option *)
	qb82KF1_4_Miscellaneous_STL						AT %Q*: BOOL;	(* Option *)
	qb82KF1_8_Spare			 						AT %Q*: BOOL;

	(*TERMINAL 83KF1 (EL2008 8Ch. Dig. Output 24V, 0.5A) ******************************************************)
	qb83KF1_1_Spare									AT %Q*: BOOL;
	qb83KF1_5_Spare									AT %Q*: BOOL;
	qb83KF1_2_Spare									AT %Q*: BOOL;
	qb83KF1_6_Spare									AT %Q*: BOOL;
	qb83KF1_3_Spare									AT %Q*: BOOL;
	qb83KF1_7_Spare									AT %Q*: BOOL;
	qb83KF1_4_Spare									AT %Q*: BOOL;
	qb83KF1_8_Spare			 						AT %Q*: BOOL;

	(*TERMINAL 90KF1 (EL2624 4Ch. Relay Output, 125 V AC, 30 V DC, 0.5 A AC, 2 A DC)******************)
	qb90KF1_1_PrintingEnableSignal						AT %Q*: BOOL;		(*M-Series Print*)
	qb90KF1_2_AlarmQuiteSignal							AT %Q*: BOOL;		(*M-Series Reset*)
	qb90KF1_3_ProductDetectSignal						AT %Q*: BOOL;		(*M-Series Apply*)
	qb90KF1_4_Spare										AT %Q*: BOOL;


	(*TERMINAL 97KF1 - EL6631 -  PROFINET IO Controller ********************************************************)
	ist97KF1_Master01PNetState 						AT %I* : ST_CX_EtherCATMasterPNetState;

	(*DRIVE  3T1  - G120C ************************************************************************************)
	ist3T1_outerseparation							AT %I* : ST_DRIVE_INPUT;
	qst3T1_outerseparation							AT %Q* : ST_DRIVE_OUTPUT;

	(*DRIVE  4T1  - G120C ************************************************************************************)
	ist4T1_transferconveyor							AT %I* : ST_DRIVE_INPUT;
	qst4T1_transferconveyor							AT %Q* : ST_DRIVE_OUTPUT;

	(*DRIVE  5T1  - G120C ************************************************************************************)
	ist5T1_outfeedconveyor							AT %I* : ST_DRIVE_INPUT;
	qst5T1_outfeedconveyor							AT %Q* : ST_DRIVE_OUTPUT;

	(*DRIVE  6T1  - G120C ************************************************************************************)
	ist6T1_additionalconveyor						AT %I* : ST_DRIVE_INPUT;
	qst6T1_additionalconveyor					AT %Q* : ST_DRIVE_OUTPUT;
END_VAR

// ---- GVLs/Global Variables/InputsOutputs_SFLX/IOVariablesEUCA_SFLX.TcGVL
{attribute 'Tc2GvlVarNames'}
VAR_GLOBAL

(*TERMINAL XXXKF1 - EK1100 **********************************************************)

(*ENCODER 333P2 - SICK AFS60A  ******************************************************)
	in333P2_PositionValue						AT %I* : UDINT;
	in333P2_RawPositionValue					AT %I* : UDINT;
	in333P2_AlarmStatus							AT %I* : UINT;
	in333P2_WarningStatus						AT %I* : UINT;

(*TERMINAL 349KF1 - EL4002 ******************************************************)
	qn349KF1_1_LightingIntensityTop						AT %Q* : INT;
	qn349KF1_2_LightingIntensityBottom					AT %Q* : INT;

(*TERMINAL 350KF1 (EL6001 Interface (RS232))  ********1-Channel Serial Interface RS232***********************)
	ib350A1_EL6001PortNo								AT %I* :  UINT;
	ist350A1_HandScannerCOMPortDataIn					AT %I* :  EL6InData22B;
	qst350A1_HandScannerCOMPortDataOut					AT %Q*: EL6OutData22B;

(*TERMINAL 351KF1 - EL4002 ******************************************************)
	qn351KF1_1_OuterValidationLightingIntensity						AT %Q* : INT;
	qn351KF1_2_OuterAggregationLightingIntensity				AT %Q* : INT;

(*TERMINAL 352KF1 - EL4002 ******************************************************)
	qn352KF1_1_CaseContentValidationLightingIntensity		AT %Q* : INT;
	qn352KF1_2_LightingIntensity							AT %Q* : INT;

(*TERMINAL 360KF1 - EL1008 ***********************************************************)
	ib360KF1_1_OuterAtInfeed							AT %I* : BOOL;	(* Option *)
	ib360KF1_5_OuterInfeedBlocked						AT %I* : BOOL;	(* Option *)
	ib360KF1_2_OuterAtLabeller							AT %I* : BOOL;
	ib360KF1_6_PackConfirmationCameraTrigSensor			AT %I* : BOOL;
	ib360KF1_3_OuterMasterListTrigSensor 					AT %I* : BOOL;
	ib360KF1_7_OuterAtReject							AT %I* : BOOL;
	ib360KF1_4_RejectConfirmation						AT %I* : BOOL;
	ib360KF1_8_RejectBinFull								AT %I* : BOOL;

(*TERMINAL 361KF1 - EL1008 ***********************************************************)
	ib361KF1_1_OuterGateExtended							AT %I* : BOOL;
	ib361KF1_5_OuterGateRetracted					AT %I* : BOOL;
	ib361KF1_2_FirstPusherExtended						AT %I* : BOOL;
	ib361KF1_6_FirstPusherRetracted						AT %I* : BOOL;
	ib361KF1_3_RejectCylinderExtended					AT %I* : BOOL;
	ib361KF1_7_RejectCylinderRetracted					AT %I* : BOOL;
	ib361KF1_4_SecondPusherExtended						AT %I* : BOOL;	(* Option *)
	ib361KF1_8_SecondPusherRetracted						AT %I* : BOOL;

(*TERMINAL 362KF1 - EL1008 ************************************************************)
	ib362KF1_1_Labeller01Ready							AT %I*: BOOL;
	ib362KF1_5_Labeller01DataReady						AT %I*: BOOL;
	ib362KF1_2_Labeller01ApplicatorHomePosition 			AT %I*: BOOL;
	ib362KF1_6_Labeller01LabelPrinted						AT %I*: BOOL;
	ib362KF1_3_Labeller01SummaryWarning					AT %I*: BOOL;
	ib362KF1_7_Labeller01Error							AT %I*: BOOL;
	ib362KF1_4_AirPressureOK							AT %I*: BOOL;
	ib362KF1_8_Labeller01InPosition					AT %I*: BOOL;	(* ??? *)

(*TERMINAL 363KF1 (EL1008 8Ch. Dig. Input 24V, 3ms) ***************************************)
	ib363KF1_1_QAButtonRejectOuter						AT %I*: BOOL;	(* Option *)
	ib363KF1_5_IntermediatePushSensor					AT %I*: BOOL;
	ib363KF1_2_CaseLabelValidationCameraTrigSensor	AT %I*: BOOL;
	ib363KF1_6_CaseAtRejectStation						AT %I*: BOOL;	(* Option *)
	ib363KF1_3_RowCompleteSensor						AT %I*: BOOL;
	ib363KF1_7_LayerCompleteSensor						AT %I*: BOOL;
	ib363KF1_4_CaseCompleteSensor						AT %I*: BOOL;
	ib363KF1_8_CaseDischargedSensor						AT %I*: BOOL;

(*TERMINAL 364KF1 (EL1008 8Ch. Dig. Input 24V, 3ms) ****************************************)
	ib364KF1_1_AdditionalRejectCylExtended				AT %I*: BOOL;
	ib364KF1_5_AdditionalRejectCylRetracted				AT %I*: BOOL;
	ib364KF1_2_OuterInfeedJam							AT %I*: BOOL;
	ib364KF1_6_PackAggregationCameraRigTrigger		AT %I*: BOOL;
	ib364KF1_3_OuterAtSideFlexExit						AT %I*: BOOL;
	ib364KF1_7_OuterTransferConfirmation				AT %I*: BOOL;
	ib364KF1_4_EUCAExitBlocked								AT %I*: BOOL;
	ib364KF1_8_EUCABuildBack							AT %I*: BOOL;

(*TERMINAL 365KF1 (EL1008 8Ch. Dig. Input 24V, 3ms) ****************************************)
	ib365KF1_1_OuterAtPostMachineInfeed				AT %I*: BOOL;
	ib365KF1_5_RejectConfirmationNCW				AT %I*: BOOL;
	ib365KF1_2_RejectBinFullNCW						AT %I*: BOOL;
	ib365KF1_6_OuterReadingConfirmation			AT %I*: BOOL;
	ib365KF1_3_OuterAtTransferReject				AT %I*: BOOL;
	ib365KF1_7_Spare									AT %I*: BOOL;
	ib365KF1_4_Spare									AT %I*: BOOL;
	ib365KF1_8_Spare									AT %I*: BOOL;

(*TERMINAL 366KF1 (EL1008 8Ch. Dig. Input 24V, 3ms) ****************************************)
	ib366KF1_1_Spare									AT %I*: BOOL;
	ib366KF1_5_Spare									AT %I*: BOOL;
	ib366KF1_2_Spare									AT %I*: BOOL;
	ib366KF1_6_Spare									AT %I*: BOOL;
	ib366KF1_3_Spare									AT %I*: BOOL;
	ib366KF1_7_Spare									AT %I*: BOOL;
	ib366KF1_4_Spare									AT %I*: BOOL;
	ib366KF1_8_Spare									AT %I*: BOOL;

(*TERMINAL 380KF1 - EL2008 (EL2008 8Ch. Dig. Output 24V, 0.5A) ********************************)
	qb380KF1_1_FirstPusherCylinderExtend				AT %Q*: BOOL;
	qb380KF1_5_SecondPusherCylinderExtend	 			AT %Q*: BOOL;
	qb380KF1_2_GateCylinderExtend 						AT %Q*: BOOL;		(*Additional reject acturator for SFLX*)
	qb380KF1_6_GateCylinderRetract	 					AT %Q*: BOOL;		(*Additional reject acturator for SFLX*)
	qb380KF1_3_RejectCylinderExtend						AT %Q*: BOOL;
	qb380KF1_7_RejectCylinderRetract			  		AT %Q*: BOOL;
	qb380KF1_4_FirstPusherCylinderRetract				AT %Q*: BOOL;
	qb380KF1_8_SecondPusherCylinderRetract				AT %Q*: BOOL;

(*TERMINAL 381KF1 (EL2008 8Ch. Dig. Output 24V, 0.5A) ***************************************)
	qb381KF1_1_RearConfirmationCameraTrigger			AT %Q*: BOOL;
	qb381KF1_5_RearConfirmationCameraPower				AT %Q*: BOOL;
	qb381KF1_2_FrontConfirmationCameraTrigger			AT %Q*: BOOL;
	qb381KF1_6_FrontConfirmationCameraPower	 			AT %Q*: BOOL;
	qb381KF1_3_OuterValidationCameraTrig 					AT %Q*: BOOL;
	qb381KF1_7_OuterValidationCameraPower				AT %Q*: BOOL;
	qb381KF1_4_OuterAggregationCameraTrig					AT %Q*: BOOL;
	qb381KF1_8_OuterAggregationCameraPower					AT %Q*: BOOL;

(*TERMINAL 382KF1 (EL2008 8Ch. Dig. Output 24V, 0.5A) ****************************************)
	qb382KF1_1_CaseContentValidationCameraTrig				AT %Q*: BOOL;
	qb382KF1_5_CaseContentValidationCameraPower			AT %Q*: BOOL;
	qb382KF1_2_CaseLabelValidationCameraTrig				AT %Q*: BOOL;
	qb382KF1_6_CaseLabelValidationCameraPower	 			AT %Q*: BOOL;
	qb382KF1_3_PackAggregationCamera1Trigger			AT %Q*: BOOL;		(*Used for SFLX*)
	qb382KF1_7_PackAggregationCamera1Power				AT %Q*: BOOL;		(*Used for SFLX*)
	qb382KF1_4_PackAggregationCamera2Trigger			AT %Q*: BOOL;		(*Used for SFLX*)
	qb382KF1_8_PackAggregationCamera2Power				AT %Q*: BOOL;		(*Used for SFLX*)

(*TERMINAL 383KF1 (EL2008 8Ch. Dig. Output 24V, 0.5A) ****************************************)
	qb383KF1_1_LightPoleGREEN						AT %Q*: BOOL;
	qb383KF1_5_LightPoleAMBER						AT %Q*: BOOL;
	qb383KF1_2_LightPoleRED						AT %Q*: BOOL;
	qb383KF1_6_LightPoleALARM						AT %Q*: BOOL;
	qb383KF1_3_OuterContentValidationCameraTrig			AT %Q*: BOOL;
	qb383KF1_7_OuterContentValidationCameraPower	AT %Q*: BOOL;
	qb383KF1_4_RejectActiveNCW										AT %Q*: BOOL;
	qb383KF1_8_Spare									AT %Q*: BOOL;

(*TERMINAL 384KF1 (EL2008 8Ch. Dig. Output 24V, 0.5A) ****************************************)
	qb384KF1_1_Spare										AT %Q*: BOOL;
	qb384KF1_5_Spare										AT %Q*: BOOL;
	qb384KF1_2_Spare										AT %Q*: BOOL;
	qb384KF1_6_Spare										AT %Q*: BOOL;
	qb384KF1_3_PLCControlledOuterValidCamLightning		AT %Q*: BOOL;
	qb384KF1_7_PLCControlledOuterAggCamLightning		AT %Q*: BOOL;
	qb384KF1_4_PLCControlledCaseContentCamLightning	AT %Q*: BOOL;
	qb384KF1_8_Spare									AT %Q*: BOOL;

(*TERMINAL 390KF1 (EL2624 4Ch. Relay Output, 125 V AC, 30 V DC, 0.5 A AC, 2 A DC)******************)
	qb390KF1_1_Labeller1ResetSignal						AT %Q*: BOOL;
	qb390KF1_2_Labeller1PrintSignal						AT %Q*: BOOL;
	qb390KF1_3_Labeller1ApplySignal						AT %Q*: BOOL;
	qb390KF1_4_DoorGuardOK								AT %Q*: BOOL;

END_VAR

// ---- GVLs/Global Variables/InputsOutputs_SFLX/IOVariablesPAOL_SFLX.TcGVL
{attribute 'Tc2GvlVarNames'}
VAR_GLOBAL

(*TERMINAL XXXKF1 - EK1100 ******************************************************)

(*TERMINAL 647KF1 - EL4002 ******************************************************)
	qn647KF1_1_LightingIntensity							AT %Q* : INT;
	qn647KF1_2_Spare									AT %Q* : INT;

(*TERMINAL 660KF1 - EL1008 ******************************************************)
	ib660KF1_1_PackAggregationCameraRigTrigger			AT %I* : BOOL;
	ib660KF1_5_PackAggregationCamera1Trigger				AT %I* : BOOL;
	ib660KF1_2_PackAggregationCamera2Trigger				AT %I* : BOOL;
	ib660KF1_6_PackAggregationCamera3Trigger				AT %I* : BOOL;
	ib660KF1_3_PreMachineBuildBack						AT %I* : BOOL;
	ib660KF1_7_TPDExitBlock								AT %I* : BOOL;
	ib660KF1_4_PackAggregationCamera4Trigger				AT %I* : BOOL;	(* Option *)
	ib660KF1_8_PackIsolatorDrive							AT %I* : BOOL;

(*TERMINAL 680KF1 - EL2008 ******************************************************)
	qb680KF1_1_PackAggregationCamera1Enable				AT %Q* : BOOL;
	qb680KF1_5_PackAggregationCamera2Enable				AT %Q* : BOOL;
	qb680KF1_2_PackAggregationCamera3Enable				AT %Q* : BOOL;
	qb680KF1_6_PackAggregationCamera1Power				AT %Q* : BOOL;
	qb680KF1_3_PackAggregationCamera2Power				AT %Q* : BOOL;
	qb680KF1_7_PackAggregationCamera3Power				AT %Q* : BOOL;
	qb680KF1_4_PackAggregationCamera4Enable				AT %Q* : BOOL;
	qb680KF1_8_PackCamerasLenseAir						AT %Q* : BOOL;

END_VAR

// ---- GVLs/Global Variables/InputsOutputs_SFLX/IOVariablesPLAS_SFLX.TcGVL
{attribute 'Tc2GvlVarNames'}
VAR_GLOBAL

(*TERMINAL XXXKF1 - EK1100 ******************************************************)

(*TERMINAL 649KF1 - EL4002 ******************************************************)
	qn649KF1_1_PackAggregationLightingIntensity				AT %Q* : INT;
	qn649KF1_2_LightingIntensity								AT %Q* : INT;

(*TERMINAL 663KF1 - EL1008 ******************************************************)
	ib663KF1_1_MasterListCameraTrigSensor					AT %I* : BOOL;
	ib663KF1_5_SpareMasterListCameraTrigSensor			AT %I* : BOOL;		(* Option *)
	ib663KF1_2_AggregationCameraTrigSensor				AT %I* : BOOL;
	ib663KF1_6_SpareAggregationCamera1TrigSensor		AT %I* : BOOL;		(* Option *)
	ib663KF1_3_SpareAggregationCamera2TrigSensor		AT %I* : BOOL;		(* Option *)
	ib663KF1_7_PackQueueIndex								AT %I* : BOOL; 		(* Option *)
	ib663KF1_4_StackQueueIndex								AT %I* : BOOL; 		(* Option *)
	ib663KF1_8_Spare											AT %I* : BOOL;

(*TERMINAL 664KF1 - EL1008 ******************************************************)
	ib664KF1_1_OuterIndexComplete							AT %I* : BOOL;
	ib664KF1_5_IntermediateCameraTrigSensor				AT %I* : BOOL;		(* TO DO Intemediat Camera Trigger *)
	ib664KF1_2_Guard1 										AT %I* : BOOL;
	ib664KF1_6_Guard2										AT %I* : BOOL;
	ib664KF1_3_Guard3 										AT %I* : BOOL;
	ib664KF1_7_Guard4 										AT %I* : BOOL;
	ib664KF1_4_OuterBrushOpen								AT %I* : BOOL;
	ib664KF1_8_RejectTowerActive							AT %I* : BOOL;

(*TERMINAL 665KF1 (EL1008 8Ch. Dig. Input 24V, 3ms) ******************************************************)
	ib665KF1_1_FilmInPosition 								AT %I*: BOOL;
	ib665KF1_5_IntermediatePrinterTrigger					AT %I*: BOOL;
	ib665KF1_2_Spare									AT %I*: BOOL;
	ib665KF1_6_Spare									AT %I*: BOOL;
	ib665KF1_3_Spare 								AT %I*: BOOL;
	ib665KF1_7_Spare									AT %I*: BOOL;
	ib665KF1_4_Spare									AT %I*: BOOL;
	ib665KF1_8_Spare 	 							AT %I*: BOOL;

(*TERMINAL 683KF1 - EL2008 ******************************************************)
	qb683KF1_1_MasterListCameraPower						AT %Q* : BOOL;
	qb683KF1_5_SpareMasterListCameraPower				AT %Q* : BOOL;	(* Option *)
	qb683KF1_2_SpareAggregationCameraPower				AT %Q* : BOOL;	(* Option *)
	qb683KF1_6_AggregationCamera1Power					AT %Q* : BOOL;
	qb683KF1_3_AggregationCamera2Power					AT %Q* : BOOL;
	qb683KF1_7_ConfirmationCamera1Power					AT %Q* : BOOL; 	(* Option *)
	qb683KF1_4_ConfirmationCamera2Power					AT %Q* : BOOL; 	(* Option *)
	qb683KF1_8_PLCControlledPackAggCamLightning		AT %Q* : BOOL;

(*TERMINAL 684KF1 - EL2008 ******************************************************)
	qb684KF1_1_MasterListCameraTrigger					AT %Q* : BOOL;
	qb684KF1_5_SpareMasterListCameraTrigger				AT %Q* : BOOL;	(* Option *)
	qb684KF1_2_AggregationCameraTrigger					AT %Q* : BOOL;
	qb684KF1_6_SpareAggregationCamera1Trigger			AT %Q* : BOOL; 	(* Option *)
	qb684KF1_3_SpareAggregationCamera2Trigger			AT %Q* : BOOL; 	(* Option *)
	qb684KF1_7_ConfirmationCamera1Trigger				AT %Q* : BOOL; 	(* Option *)
	qb684KF1_4_ConfirmationCamera2Trigger				AT %Q* : BOOL; 	(* Option *)
	qb684KF1_8_Spare											AT %Q* : BOOL;

(*TERMINAL 685KF1 (EL2008 8Ch. Dig. Output 24V, 3ms) ******************************************************)
	qb685KF1_1_IntermediateCameraTrigger								AT %Q*: BOOL;
	qb685KF1_5_IntermediateCameraPower									AT %Q*: BOOL;
	qb685KF1_2_Spare									AT %Q*: BOOL;
	qb685KF1_6_Spare									AT %Q*: BOOL;
	qb685KF1_3_Spare								AT %Q*: BOOL;
	qb685KF1_7_Spare								AT %Q*: BOOL;
	qb685KF1_4_Spare										AT %Q*: BOOL;
	qb685KF1_8_Spare 							AT %Q*: BOOL;

END_VAR

// ---- GVLs/Global Variables/_VERSION/_VERSION_CONTROL.TcGVL
{attribute 'Tc2GvlVarNames'}
VAR_GLOBAL
	(*cRELEASE_DATE		: STRING[10] := '25.03.2025';*)

	cHARDWARE_CONFIG_VERSION	: STRING[20] := 'IND-METS-NCW_v007';
	(*cVERSION_INFO		: T_MaxString := '26/07/23 - 07.00.41 - SD - UPS management';*)
END_VAR

(*
Version history:

Date		|	Version/Author 		|	Remark
----------------------------------------------------------------------------------------------------
26/07/23	|	07.00.41	SD		|	UPS management and power related Alarm and Warnings
25/07/23	|	07.00.40	SD		|	UPS management draft
19/07/23	|	07.00.39	SD		|	PLAS sequence placeholder
18/07/23	|	07.00.38	TW SD	|	Hand scsnner selection mod
09/05/23	|	07.00.02	PP		|	Add remaining HotFixes form Korea (according Jira tasks)
			|						|	
09/11/22	|	06.37.05	PP		|	Add Log system for case level (EventCT) and VERSION_CONTROL
05/11/22	|	06.37.03	PP		|	Original PLC-METS-6.37.03_Inline.pro from Piotr
15/09/22	|	06.37.01	PP		|	Lateste hardware design implemented HC METS-INLINE v2.10
*)

// ---- Version/Global_Version.TcGVL
{attribute 'TcGenerated'}
{attribute 'no-analysis'}
{attribute 'linkalways'}
// This function has been automatically generated from the project information.
VAR_GLOBAL CONSTANT
	{attribute 'const_non_replaced'}
	stLibVersion_AlarmsHandler : ST_LibVersion := (iMajor := 1, iMinor := 0, iBuild := 0, iRevision := 0, nFlags := 0, sVersion := '1.0.0.0');
END_VAR

// ---- POUs/Alarm/F_ALARM_SetDefinition.TcPOU
(*Max text message cannot exceed 255 char including perfedeined: ('MessageTypeNo:=', INT_TO_STRING(nMessageTypeNo), ' ; MessageInfo="',sTextMessage,'"', ' ; AutoReset=', BOOL_TO_STRING(bAutoReset))*)
FUNCTION F_ALARM_SetDefinition : BOOL
VAR_INPUT
	bAlarmTrigger 				: BOOL;
	nCategoryNo				: INT;
	nMessageTypeNo			: INT;
	sTextMessage				: STRING(200); (* Number of 200 char + 51 char form predefined message*)
	tAlarmTimout 				: TIME :=t#1000ms;
	bAlarmDefinitionEnable 	: BOOL;
	bInhibitReset 				: BOOL;
//	bInternalReset 				: BOOL;
END_VAR

VAR
	sMessagePrfix				: T_Char;
	sMessageNo				: STRING(3);

	bAutoReset 				: BOOL;
	nGroupIndex 				: INT;
	nActualAlarmPosition		: INT;
END_VAR
(*All VAR_IN_OUT variables have been moved to the end of the declaration due to compatibility reasons*)
VAR_IN_OUT
	aAlarmsSettings 		: ARRAY [0..cMAX_ALARM_GROUP] OF ST_AlarmSettings;
	nAlarmIndex				: INT;
	sMsgInfo				: T_MaxString;
	stMsgAux				: ST_ALARM_Aux;
END_VAR

nAlarmIndex := LIMIT(0, nAlarmIndex, cMAX_MESSAGE_NUMBER);

//**********************************************************************************************************	

IF nAlarmIndex <> cMAX_MESSAGE_NUMBER THEN

	nGroupIndex:= nAlarmIndex/32;
	nActualAlarmPosition:= nAlarmIndex MOD 32;
	
	IF nMessageTypeNo >= 0  AND  nMessageTypeNo <= 15 THEN

		sMessagePrfix := 'A';
		IF nMessageTypeNo > 7 THEN; 	(*Message type from 8 to 15 are set up as warrninrg*)
			bAutoReset 		:= TRUE;
			sMessagePrfix 	:= 'W';
		END_IF

		sMessageNo := F_AddPadding(nAlarmIndex, 3);

		IF NOT bAlarmDefinitionEnable THEN
			
			sTextMessage :=  F_CONCAT5('(','D',sMessageNo,') ','ALARM MANAGEMENT BLOCK DISABLE');
		ELSIF sTextMessage = '' THEN

			sTextMessage :=  F_CONCAT5('(','S',sMessageNo,') ','ALARM MISSING DESCRIPTION');
		ELSE
			
			sTextMessage :=  F_CONCAT5('(',sMessagePrfix,sMessageNo,') ',sTextMessage);
		END_IF
	
		IF stMsgAux.bAutoReset <> bAutoReset OR stMsgAux.nCategoryNo <> nCategoryNo OR stMsgAux.nMessageTypeNo <> nMessageTypeNo OR stMsgAux.sTextMessage <> sTextMessage THEN

			sMsgInfo := F_CONCAT9('Cat=',INT_TO_STRING(nCategoryNo),';MsgType=', INT_TO_STRING(nMessageTypeNo),';MsgInfo="',sTextMessage,'"', ';AutoRst=', BOOL_TO_STRING(bAutoReset));
		END_IF

		aAlarmsSettings[nGroupIndex].aTextMessageTable[nActualAlarmPosition]		:= sTextMessage;
		aAlarmsSettings[nGroupIndex].aAlarmTriggerTable[nActualAlarmPosition]		:= bAlarmTrigger ;
		aAlarmsSettings[nGroupIndex].aAlarmTimoutTable[nActualAlarmPosition]		:= tAlarmTimout;
		aAlarmsSettings[nGroupIndex].aBlockEnableTable[nActualAlarmPosition]		:= bAlarmDefinitionEnable;
		aAlarmsSettings[nGroupIndex].aInhibitResetTable[nActualAlarmPosition]		:= bInhibitReset AND bAlarmDefinitionEnable;
		aAlarmsSettings[nGroupIndex].aAutoResetTable[nActualAlarmPosition]			:= bAutoReset;
		aAlarmsSettings[nGroupIndex].aCategoryNoTable[nActualAlarmPosition]			:= nCategoryNo;
		aAlarmsSettings[nGroupIndex].aMessageTypeStatusTable[nActualAlarmPosition]	:= F_FiltredSetBitState16(TRUE, 'ALL', nMessageTypeNo, TRUE, aAlarmsSettings[nGroupIndex].aMessageTypeStatusTable[nActualAlarmPosition]);
		
	ELSE	
		sMessageNo := F_AddPadding(nAlarmIndex, 3);
		sTextMessage :=  F_CONCAT5('(','D',sMessageNo,') ','ALARM DISABLE BY WRONG MESSAGE TYPE');
		aAlarmsSettings[nGroupIndex].aTextMessageTable[nActualAlarmPosition]	:= sTextMessage;
		
		IF stMsgAux.bAutoReset <> bAutoReset OR stMsgAux.nCategoryNo <> nCategoryNo OR stMsgAux.nMessageTypeNo <> nMessageTypeNo OR stMsgAux.sTextMessage <> sTextMessage THEN

			sMsgInfo := F_CONCAT9('Cat=',INT_TO_STRING(0),';MsgType:=', INT_TO_STRING(-1),';MsgInfo="',sTextMessage,'"', ';AutoRst=', BOOL_TO_STRING(FALSE));
		END_IF
	END_IF

	nAlarmIndex := nAlarmIndex +1;
	F_ALARM_SetDefinition := TRUE;
	
ELSE
	sTextMessage :=  F_CONCAT4('(','D255',') ','ALARM NUMBER MAX LIMIT');
	aAlarmsSettings[7].aTextMessageTable[31]	:= sTextMessage;
	
	IF stMsgAux.bAutoReset <> bAutoReset OR stMsgAux.nCategoryNo <> nCategoryNo OR stMsgAux.nMessageTypeNo <> nMessageTypeNo OR stMsgAux.sTextMessage <> sTextMessage THEN

		sMsgInfo := F_CONCAT9('Cat=',INT_TO_STRING(0),';MsgType:=', INT_TO_STRING(-2),';MsgInfo="',sTextMessage,'"', ';AutoRst=', BOOL_TO_STRING(FALSE));
	END_IF	
END_IF

//**********************************************************************************************************	
stMsgAux.bAutoReset 	:= bAutoReset;
stMsgAux.nCategoryNo	:= nCategoryNo;
stMsgAux.nMessageTypeNo	:= nMessageTypeNo;
stMsgAux.sTextMessage	:= sTextMessage;

END_FUNCTION
